(* PLC project SafeLOGIC-1, BrAutomation SafeDESIGNER 2.90.21.261 *)
(* stored: companyURL http://www.br-automation.com, creationDateTime Tue Mar 18 08:17:32 2014 *)

PROGRAM Main

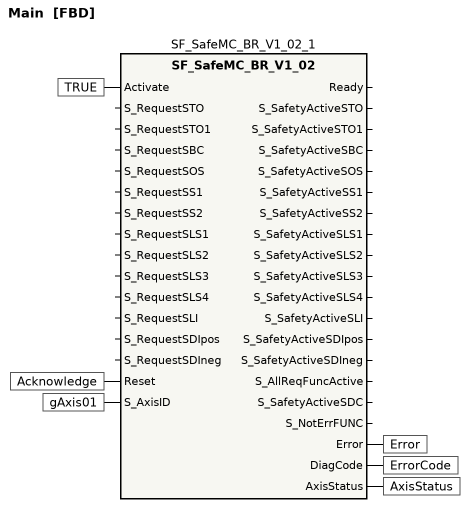
(* FBD diagram, written out as Structured Text *)
SF_SafeMC_BR_V1_02_1(Activate := TRUE, Reset := Acknowledge, S_AxisID := gAxis01);
Error := SF_SafeMC_BR_V1_02_1.Error;
ErrorCode := SF_SafeMC_BR_V1_02_1.DiagCode;
AxisStatus := SF_SafeMC_BR_V1_02_1.AxisStatus;
END_PROGRAM
